INTERFACE I_MaterialSection

METHOD changeRobotsEOAT : BOOL
VAR_INPUT
END_VAR
END_METHOD

METHOD load : BOOL
VAR_INPUT
	pair : REFERENCE TO PositionMaterials;
END_VAR
END_METHOD

METHOD unload : BOOL
VAR_INPUT
END_VAR
END_METHOD

METHOD usesMaterial : BOOL
VAR_INPUT
END_VAR
END_METHOD

END_INTERFACE

(* stored: Version 1.1.0.1, ProductVersion 3.1.4024.11
   Itf I_MaterialSection: Id {60a8100d-09a1-43bb-843f-e7486ceeed19}
   Method changeRobotsEOAT: Id {63d8ef9d-f8aa-4c79-af4b-d53b87a37256}
   Method load: Id {7d7921c2-22d8-4c27-b548-abfae784bce2}
   Method unload: Id {84095436-e4a6-4f8a-a0c6-e9783af45db9}
   Method usesMaterial: Id {a5fca9bb-eb53-4844-8e77-c5b578cca39e} *)
